FUNCTION_BLOCK FB_VALVE_RELAY 
VAR_IN_OUT
END_VAR
VAR_INPUT
END_VAR
VAR_OUTPUT
	bTimerQ : BOOL;
END_VAR
VAR
	b_open : BOOL; // control variable
	// EL2624 Relayu Logic Here

	rawOutputRelayChan1 AT %Q*: BOOL;
	rawOutputRelayChan3 AT %Q*: BOOL;
	bCloseRBV AT %I* : BOOL;
	bOpenRBV AT %I* : BOOL;
	bMovingRBV AT %I* : BOOL;
	
	tActuateTime : TIME := T#24h;
	iState: INT;
	fbValveTimer : TON;
END_VAR


fbValveTimer(IN:=TRUE, PT:=tActuateTime);

CASE iState OF
    E_VALVE_RELAY_STATES.INIT: // INIT
    fbValveTimer(IN:=FALSE); //RESTART TIMER
    iState := E_VALVE_RELAY_STATES.NOMINAL;

    E_VALVE_RELAY_STATES.NOMINAL: // NOMINAL
	ACTUATE_VALVE(b_open); 
 
	IF fbValveTimer.Q THEN iState := E_VALVE_RELAY_STATES.ACTUATE; END_IF
	
	E_VALVE_RELAY_STATES.ACTUATE: // Do the opposite of current valve state
	IF bCloseRBV THEN ACTUATE_VALVE(TRUE);END_IF
	IF bOpenRBV THEN ACTUATE_VALVE(FALSE);END_IF
	IF bMovingRBV THEN iState := E_VALVE_RELAY_STATES.WAIT; END_IF; // Only transition when we have started to move
	
	E_VALVE_RELAY_STATES.WAIT: // Go back to init to reset timer and return valve to previous state.
	IF NOT bMovingRBV THEN iState := E_VALVE_RELAY_STATES.INIT; END_IF;

END_CASE

bTimerQ := fbValveTimer.Q;

METHOD ACTUATE_VALVE : BOOL
VAR_INPUT
	b_open: BOOL;
END_VAR
IF b_open THEN
	rawOutputRelayChan1 := FALSE;
	rawOutputRelayChan3 := TRUE;
ELSE
	rawOutputRelayChan1 := TRUE;
	rawOutputRelayChan3 := FALSE;
END_IF
END_METHOD

END_FUNCTION_BLOCK

(* stored: Version 1.1.0.1, ProductVersion 3.1.4024.11
   POU FB_VALVE_RELAY: Id {e2531ff2-ea72-4542-bd8f-7299f2dc48b9}, SpecialFunc None
   Method ACTUATE_VALVE: Id {919e3d16-476c-4acf-ad5c-4fabd5d630e2} *)
